{attribute addProperty BoxType "EL2252--0000"}
{attribute addProperty Id "ActivateAT %Q*USINT81"}
{attribute addProperty CRC "62507382"}
{attribute addProperty SizeInBites "8"}
{attribute addProperty SizeInBytes "1"}
TYPE DC_Sync_Activate_03B9C976 :
STRUCT
	{attribute addProperty Name "Activate"}
	Activate AT %Q* : USINT;
END_STRUCT
END_TYPE

(* stored: Version 1.2.0.0, ProductVersion 3.1.4024.9
   DUT DC_Sync_Activate_03B9C976: Id {4cbfa084-33aa-4863-a141-a7b898c22955} *)
